// TIA Portal V17 export
// export: Created 2025-03-07T09:19:10.1766276Z, ExportSetting WithDefaults, DisplayName Totally Integrated Automation Portal, DisplayVersion V17 Update 8, DisplayName TIA Portal Openness, DisplayVersion V17 Update 8, DisplayName TIA Portal Version Control Interface, DisplayVersion V17, DisplayName SINAMICS Startdrive Advanced, DisplayVersion V17 SP2, DisplayName SINAMICS Startdrive G110M, G120, G120C, G120D, G120P, G115D, DisplayVersion V17 SP2, DisplayName SINAMICS Startdrive G130, G150, S120, S150, SINAMICS MV, S210, DisplayVersion V17 SP2, DisplayName STEP 7 Professional, DisplayVersion V17 Update 8, DisplayName SINUMERIK ONE STEP 7 Toolbox, DisplayVersion V17 Update 12, DisplayName SINUMERIK 840D sl STEP 7 Toolbox, DisplayVersion V17 Update 12, DisplayName STEP 7 Safety, DisplayVersion V17 Update 6, DisplayName WinCC Advanced, DisplayVersion V17 Update 8
FUNCTION "FC7216_RECIPES" : Void   // FC7216, LAD
{ S7_Optimized_Access := 'FALSE' }
AUTHOR : ETXETAR
VERSION : 1.0
// stored: AutoNumber false, IsIECCheckEnabled false, SetENOAutomatically false, UDAEnableTagReadback false
   VAR_TEMP
      STRING_AUX : String[254];
      TEMP0 : Int;
      NUM_OF_RECIPES : Int;
   END_VAR
   VAR CONSTANT
      FC_NUMBER : DInt := 7216;
   END_VAR
   VAR_TEMP   // added for the SCL form of the ladder/FBD networks
      _w1 : Bool;
      _w2 : Bool;
      _w3 : Bool;
   END_VAR
BEGIN

REGION Network 1: SEQUENCE IN PROCESS
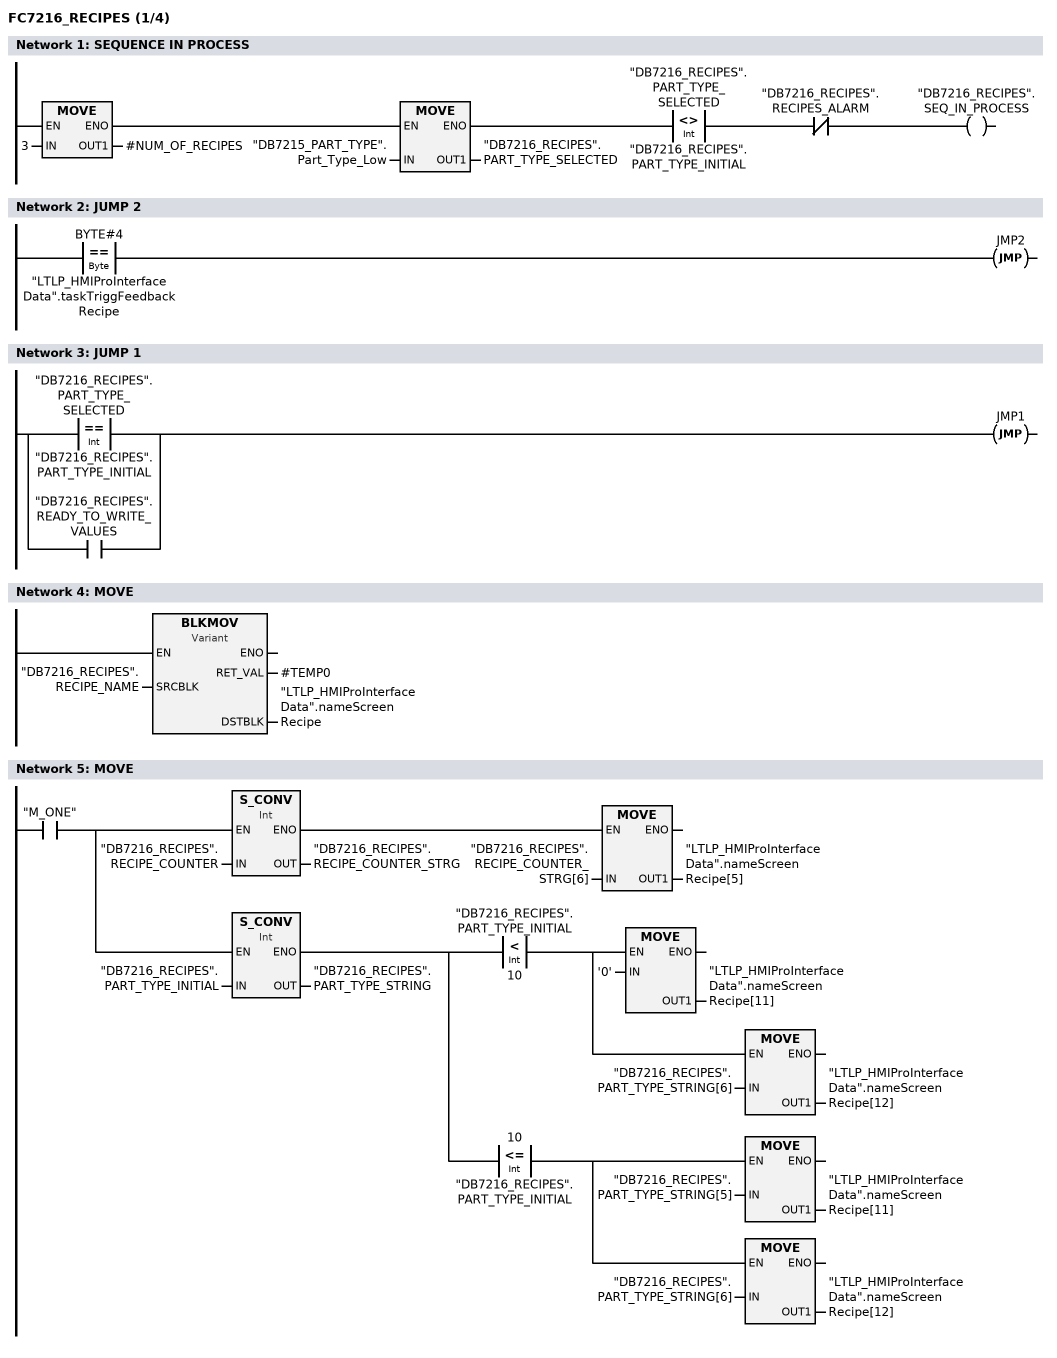
   RUNG wire#powerrail
      { S7_GenerateENO := "TRUE" } Move(in := 3, out1 => #NUM_OF_RECIPES)
      { S7_GenerateENO := "TRUE" } Move(in := "DB7215_PART_TYPE".Part_Type_Low, out1 => "DB7216_RECIPES".PART_TYPE_SELECTED)
      { S7_Templates := "SrcType := Int" } NE_Contact(in1 := "DB7216_RECIPES".PART_TYPE_SELECTED, in2 := "DB7216_RECIPES".PART_TYPE_INITIAL)
      I_Contact( "DB7216_RECIPES".RECIPES_ALARM )
      Coil( "DB7216_RECIPES".SEQ_IN_PROCESS )
   END_RUNG
   // the same network as SCL:
   // ENO of a box is taken as its EN; it also drops when the box reports an error
   #NUM_OF_RECIPES := 3;
   "DB7216_RECIPES".PART_TYPE_SELECTED := "DB7215_PART_TYPE".Part_Type_Low;
   "DB7216_RECIPES".SEQ_IN_PROCESS := ("DB7216_RECIPES".PART_TYPE_SELECTED <> "DB7216_RECIPES".PART_TYPE_INITIAL) AND NOT "DB7216_RECIPES".RECIPES_ALARM;
END_REGION

REGION Network 2: JUMP 2
   RUNG wire#powerrail
      { S7_Templates := "SrcType := Byte" } EQ_Contact(in1 := BYTE#4, in2 := "LTLP_HMIProInterfaceData".taskTriggFeedbackRecipe)
      JumpCoil( JMP2 )
   END_RUNG
   // the same network as SCL:
   IF BYTE#4 = "LTLP_HMIProInterfaceData".taskTriggFeedbackRecipe THEN GOTO JMP2; END_IF;
END_REGION

REGION Network 3: JUMP 1
   RUNG wire#powerrail
      { S7_Templates := "SrcType := Int" } EQ_Contact(in1 := "DB7216_RECIPES".PART_TYPE_SELECTED, in2 := "DB7216_RECIPES".PART_TYPE_INITIAL)
      wire#w1
      JumpCoil( JMP1 )
   END_RUNG
   RUNG wire#powerrail
      Contact( "DB7216_RECIPES".READY_TO_WRITE_VALUES )
   END_RUNG wire#w1
   // the same network as SCL:
   IF ("DB7216_RECIPES".PART_TYPE_SELECTED = "DB7216_RECIPES".PART_TYPE_INITIAL) OR "DB7216_RECIPES".READY_TO_WRITE_VALUES THEN
       GOTO JMP1;
   END_IF;
END_REGION

REGION Network 4: MOVE
   RUNG wire#powerrail
      { S7_Templates := "blk_type := Variant" } BLKMOV(SRCBLK := "DB7216_RECIPES".RECIPE_NAME, RET_VAL => #TEMP0, DSTBLK => "LTLP_HMIProInterfaceData".nameScreenRecipe)
   END_RUNG
   // the same network as SCL:
   #TEMP0 := BLKMOV(SRCBLK := "DB7216_RECIPES".RECIPE_NAME,
                    DSTBLK => "LTLP_HMIProInterfaceData".nameScreenRecipe);
END_REGION

REGION Network 5: MOVE
   RUNG wire#powerrail
      Contact( "M_ONE" )
      wire#w1
      { S7_Templates := "[src_type := Int, dest_type := String]" } S_CONV(IN := "DB7216_RECIPES".RECIPE_COUNTER, OUT => "DB7216_RECIPES".RECIPE_COUNTER_STRG)
      { S7_GenerateENO := "TRUE" } Move(in := "DB7216_RECIPES".RECIPE_COUNTER_STRG[6], out1 => "LTLP_HMIProInterfaceData".nameScreenRecipe[5])
   END_RUNG
   RUNG wire#w1
      { S7_Templates := "[src_type := Int, dest_type := String]" } S_CONV(IN := "DB7216_RECIPES".PART_TYPE_INITIAL, OUT => "DB7216_RECIPES".PART_TYPE_STRING)
      wire#w2
      { S7_Templates := "SrcType := Int" } LT_Contact(in1 := "DB7216_RECIPES".PART_TYPE_INITIAL, in2 := 10)
      wire#w3
      { S7_GenerateENO := "TRUE" } Move(in := '0', out1 => "LTLP_HMIProInterfaceData".nameScreenRecipe[11])
   END_RUNG
   RUNG wire#w3
      { S7_GenerateENO := "TRUE" } Move(in := "DB7216_RECIPES".PART_TYPE_STRING[6], out1 => "LTLP_HMIProInterfaceData".nameScreenRecipe[12])
   END_RUNG
   RUNG wire#w2
      { S7_Templates := "SrcType := Int" } LE_Contact(in1 := 10, in2 := "DB7216_RECIPES".PART_TYPE_INITIAL)
      wire#w4
      { S7_GenerateENO := "TRUE" } Move(in := "DB7216_RECIPES".PART_TYPE_STRING[5], out1 => "LTLP_HMIProInterfaceData".nameScreenRecipe[11])
   END_RUNG
   RUNG wire#w4
      { S7_GenerateENO := "TRUE" } Move(in := "DB7216_RECIPES".PART_TYPE_STRING[6], out1 => "LTLP_HMIProInterfaceData".nameScreenRecipe[12])
   END_RUNG
   // the same network as SCL:
   #_w2 := "M_ONE";
   S_CONV(EN := "M_ONE",
          IN := "DB7216_RECIPES".RECIPE_COUNTER,
          OUT => "DB7216_RECIPES".RECIPE_COUNTER_STRG,
          ENO => #_w1);
   IF #_w1 THEN
       "LTLP_HMIProInterfaceData".nameScreenRecipe[5] := "DB7216_RECIPES".RECIPE_COUNTER_STRG[6];
   END_IF;
   S_CONV(EN := #_w2,
          IN := "DB7216_RECIPES".PART_TYPE_INITIAL,
          OUT => "DB7216_RECIPES".PART_TYPE_STRING,
          ENO => #_w3);
   IF #_w3 AND ("DB7216_RECIPES".PART_TYPE_INITIAL < 10) THEN
       "LTLP_HMIProInterfaceData".nameScreenRecipe[11] := '0';
       "LTLP_HMIProInterfaceData".nameScreenRecipe[12] := "DB7216_RECIPES".PART_TYPE_STRING[6];
   END_IF;
   IF #_w3 AND (10 <= "DB7216_RECIPES".PART_TYPE_INITIAL) THEN
       "LTLP_HMIProInterfaceData".nameScreenRecipe[11] := "DB7216_RECIPES".PART_TYPE_STRING[5];
       "LTLP_HMIProInterfaceData".nameScreenRecipe[12] := "DB7216_RECIPES".PART_TYPE_STRING[6];
   END_IF;
END_REGION

REGION Network 6: MOVE
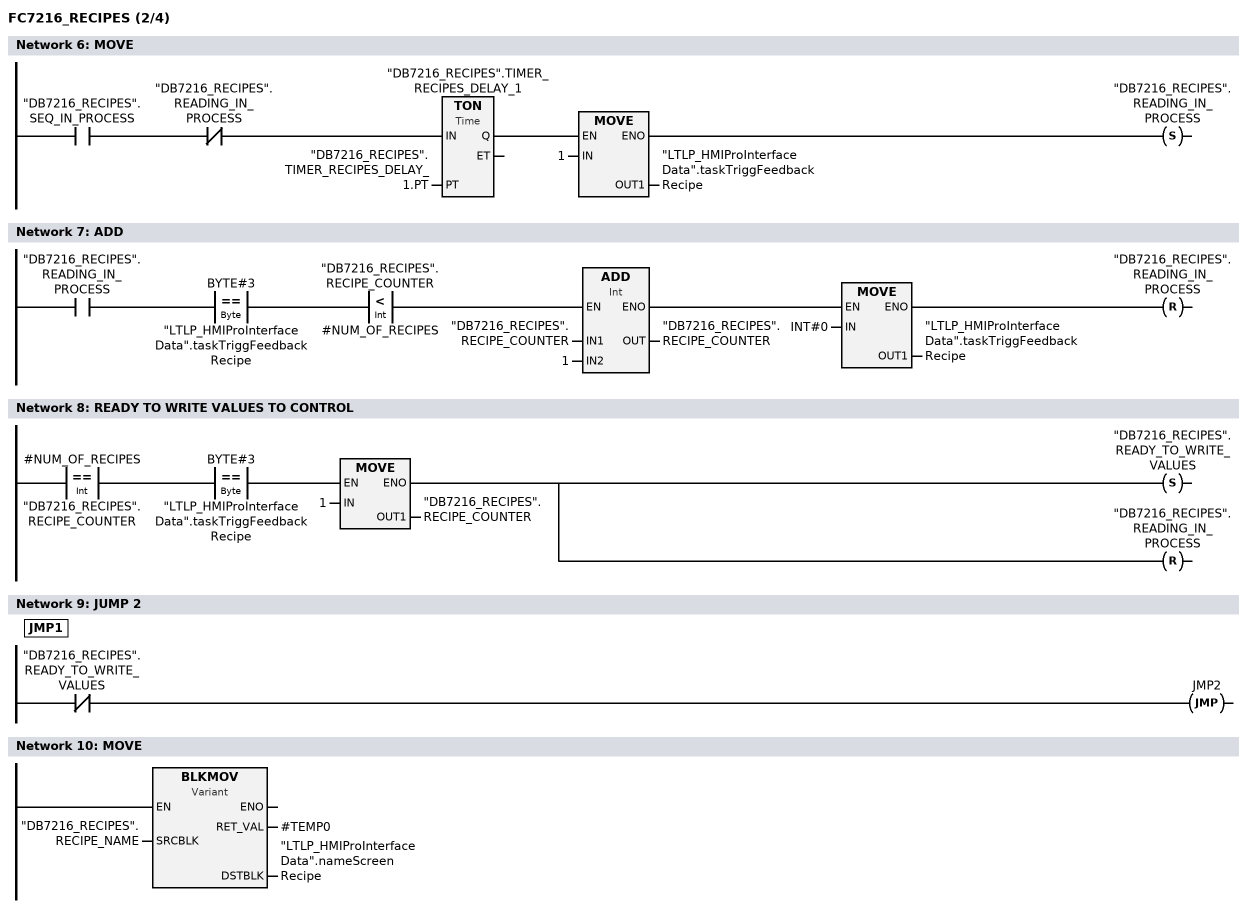
   RUNG wire#powerrail
      Contact( "DB7216_RECIPES".SEQ_IN_PROCESS )
      I_Contact( "DB7216_RECIPES".READING_IN_PROCESS )
      { S7_Templates := "time_type := Time" } "DB7216_RECIPES".TIMER_RECIPES_DELAY_1.TON(pt := "DB7216_RECIPES".TIMER_RECIPES_DELAY_1.PT, et =>)
      { S7_GenerateENO := "TRUE" } Move(in := 1, out1 => "LTLP_HMIProInterfaceData".taskTriggFeedbackRecipe)
      S_Coil( "DB7216_RECIPES".READING_IN_PROCESS )
   END_RUNG
   // the same network as SCL:
   // ENO of a box is taken as its EN; it also drops when the box reports an error
   "DB7216_RECIPES".TIMER_RECIPES_DELAY_1.TON(IN := "DB7216_RECIPES".SEQ_IN_PROCESS AND NOT "DB7216_RECIPES".READING_IN_PROCESS,
                           PT := "DB7216_RECIPES".TIMER_RECIPES_DELAY_1.PT);
   IF "DB7216_RECIPES".TIMER_RECIPES_DELAY_1.Q THEN
       "LTLP_HMIProInterfaceData".taskTriggFeedbackRecipe := 1;
       "DB7216_RECIPES".READING_IN_PROCESS := TRUE;
   END_IF;
END_REGION

REGION Network 7: ADD
   RUNG wire#powerrail
      Contact( "DB7216_RECIPES".READING_IN_PROCESS )
      { S7_Templates := "SrcType := Byte" } EQ_Contact(in1 := BYTE#3, in2 := "LTLP_HMIProInterfaceData".taskTriggFeedbackRecipe)
      { S7_Templates := "SrcType := Int" } LT_Contact(in1 := "DB7216_RECIPES".RECIPE_COUNTER, in2 := #NUM_OF_RECIPES)
      { S7_Templates := "SrcType := Int"; S7_GenerateENO := "TRUE" } Add(in1 := "DB7216_RECIPES".RECIPE_COUNTER, in2 := 1, out => "DB7216_RECIPES".RECIPE_COUNTER)
      { S7_GenerateENO := "TRUE" } Move(in := INT#0, out1 => "LTLP_HMIProInterfaceData".taskTriggFeedbackRecipe)
      R_Coil( "DB7216_RECIPES".READING_IN_PROCESS )
   END_RUNG
   // the same network as SCL:
   // ENO of a box is taken as its EN; it also drops when the box reports an error
   #_w1 := "DB7216_RECIPES".READING_IN_PROCESS AND (BYTE#3 = "LTLP_HMIProInterfaceData".taskTriggFeedbackRecipe) AND ("DB7216_RECIPES".RECIPE_COUNTER < #NUM_OF_RECIPES);
   IF #_w1 THEN
       "DB7216_RECIPES".RECIPE_COUNTER := "DB7216_RECIPES".RECIPE_COUNTER + 1;
       "LTLP_HMIProInterfaceData".taskTriggFeedbackRecipe := INT#0;
       "DB7216_RECIPES".READING_IN_PROCESS := FALSE;
   END_IF;
END_REGION

REGION Network 8: READY TO WRITE VALUES TO CONTROL
   RUNG wire#powerrail
      { S7_Templates := "SrcType := Int" } EQ_Contact(in1 := #NUM_OF_RECIPES, in2 := "DB7216_RECIPES".RECIPE_COUNTER)
      { S7_Templates := "SrcType := Byte" } EQ_Contact(in1 := BYTE#3, in2 := "LTLP_HMIProInterfaceData".taskTriggFeedbackRecipe)
      { S7_GenerateENO := "TRUE" } Move(in := 1, out1 => "DB7216_RECIPES".RECIPE_COUNTER)
      wire#w1
      S_Coil( "DB7216_RECIPES".READY_TO_WRITE_VALUES )
   END_RUNG
   RUNG wire#w1
      R_Coil( "DB7216_RECIPES".READING_IN_PROCESS )
   END_RUNG
   // the same network as SCL:
   // ENO of a box is taken as its EN; it also drops when the box reports an error
   #_w1 := (#NUM_OF_RECIPES = "DB7216_RECIPES".RECIPE_COUNTER) AND (BYTE#3 = "LTLP_HMIProInterfaceData".taskTriggFeedbackRecipe);
   IF #_w1 THEN
       "DB7216_RECIPES".RECIPE_COUNTER := 1;
       "DB7216_RECIPES".READY_TO_WRITE_VALUES := TRUE;
       "DB7216_RECIPES".READING_IN_PROCESS := FALSE;
   END_IF;
END_REGION

REGION Network 9: JUMP 2
   Label( JMP1 )
   RUNG wire#powerrail
      I_Contact( "DB7216_RECIPES".READY_TO_WRITE_VALUES )
      JumpCoil( JMP2 )
   END_RUNG
   // the same network as SCL:
   JMP1:
   IF NOT "DB7216_RECIPES".READY_TO_WRITE_VALUES THEN GOTO JMP2; END_IF;
END_REGION

REGION Network 10: MOVE
   RUNG wire#powerrail
      { S7_Templates := "blk_type := Variant" } BLKMOV(SRCBLK := "DB7216_RECIPES".RECIPE_NAME, RET_VAL => #TEMP0, DSTBLK => "LTLP_HMIProInterfaceData".nameScreenRecipe)
   END_RUNG
   // the same network as SCL:
   #TEMP0 := BLKMOV(SRCBLK := "DB7216_RECIPES".RECIPE_NAME,
                    DSTBLK => "LTLP_HMIProInterfaceData".nameScreenRecipe);
END_REGION

REGION Network 11: MOVE
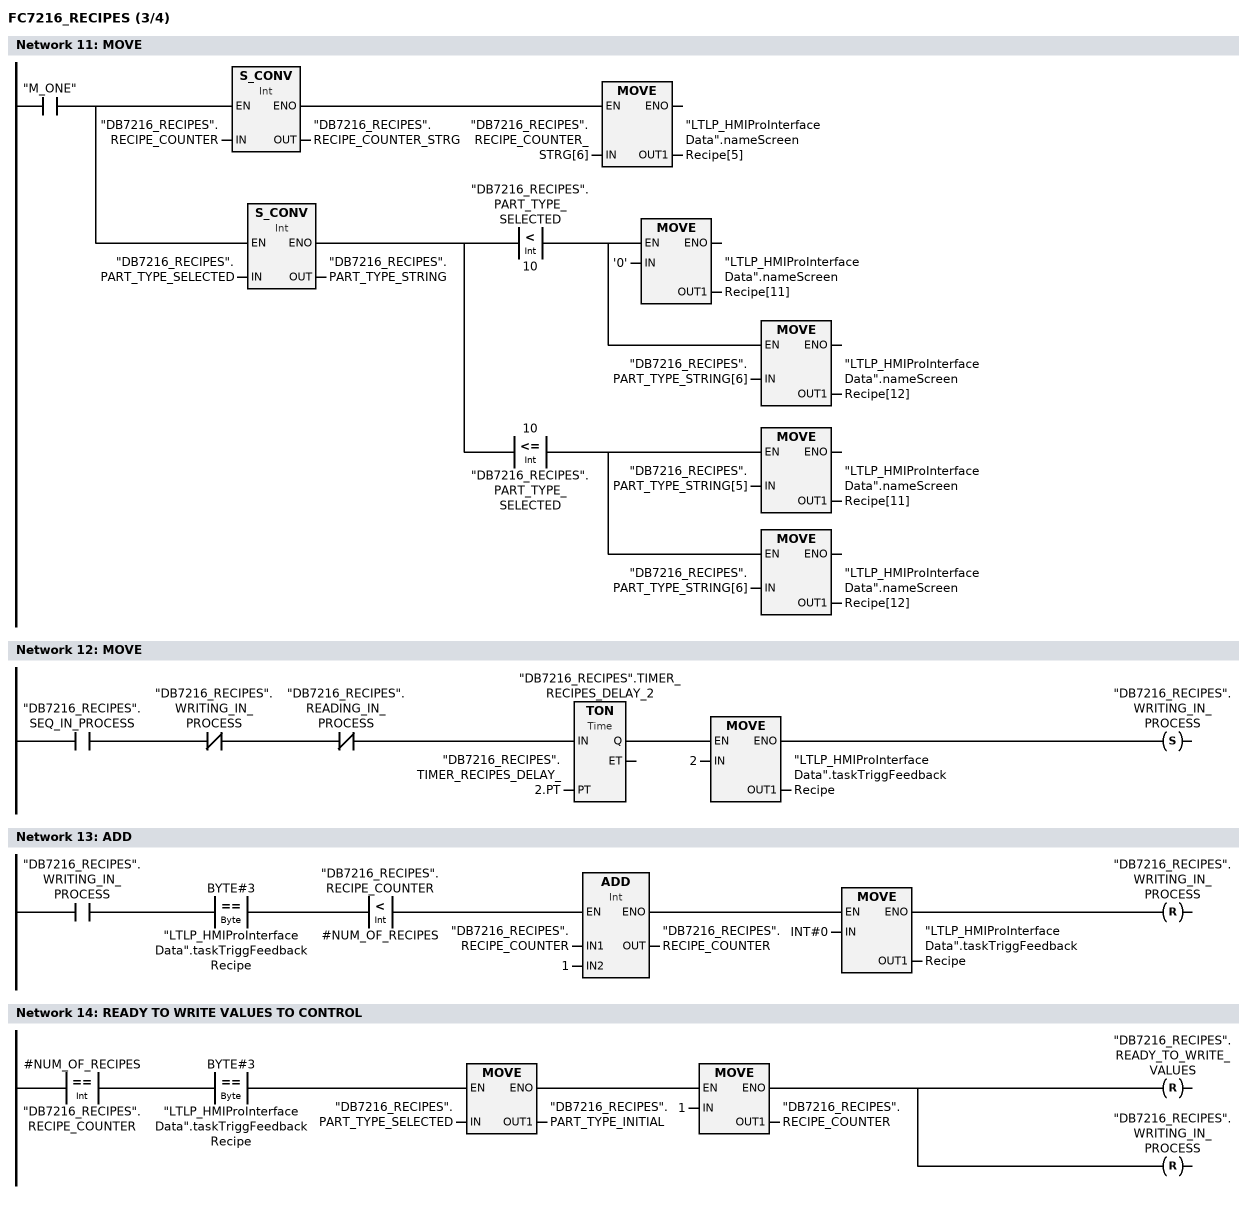
   RUNG wire#powerrail
      Contact( "M_ONE" )
      wire#w1
      { S7_Templates := "[src_type := Int, dest_type := String]" } S_CONV(IN := "DB7216_RECIPES".RECIPE_COUNTER, OUT => "DB7216_RECIPES".RECIPE_COUNTER_STRG)
      { S7_GenerateENO := "TRUE" } Move(in := "DB7216_RECIPES".RECIPE_COUNTER_STRG[6], out1 => "LTLP_HMIProInterfaceData".nameScreenRecipe[5])
   END_RUNG
   RUNG wire#w1
      { S7_Templates := "[src_type := Int, dest_type := String]" } S_CONV(IN := "DB7216_RECIPES".PART_TYPE_SELECTED, OUT => "DB7216_RECIPES".PART_TYPE_STRING)
      wire#w2
      { S7_Templates := "SrcType := Int" } LT_Contact(in1 := "DB7216_RECIPES".PART_TYPE_SELECTED, in2 := 10)
      wire#w3
      { S7_GenerateENO := "TRUE" } Move(in := '0', out1 => "LTLP_HMIProInterfaceData".nameScreenRecipe[11])
   END_RUNG
   RUNG wire#w3
      { S7_GenerateENO := "TRUE" } Move(in := "DB7216_RECIPES".PART_TYPE_STRING[6], out1 => "LTLP_HMIProInterfaceData".nameScreenRecipe[12])
   END_RUNG
   RUNG wire#w2
      { S7_Templates := "SrcType := Int" } LE_Contact(in1 := 10, in2 := "DB7216_RECIPES".PART_TYPE_SELECTED)
      wire#w4
      { S7_GenerateENO := "TRUE" } Move(in := "DB7216_RECIPES".PART_TYPE_STRING[5], out1 => "LTLP_HMIProInterfaceData".nameScreenRecipe[11])
   END_RUNG
   RUNG wire#w4
      { S7_GenerateENO := "TRUE" } Move(in := "DB7216_RECIPES".PART_TYPE_STRING[6], out1 => "LTLP_HMIProInterfaceData".nameScreenRecipe[12])
   END_RUNG
   // the same network as SCL:
   #_w2 := "M_ONE";
   S_CONV(EN := "M_ONE",
          IN := "DB7216_RECIPES".RECIPE_COUNTER,
          OUT => "DB7216_RECIPES".RECIPE_COUNTER_STRG,
          ENO => #_w1);
   IF #_w1 THEN
       "LTLP_HMIProInterfaceData".nameScreenRecipe[5] := "DB7216_RECIPES".RECIPE_COUNTER_STRG[6];
   END_IF;
   S_CONV(EN := #_w2,
          IN := "DB7216_RECIPES".PART_TYPE_SELECTED,
          OUT => "DB7216_RECIPES".PART_TYPE_STRING,
          ENO => #_w3);
   IF #_w3 AND ("DB7216_RECIPES".PART_TYPE_SELECTED < 10) THEN
       "LTLP_HMIProInterfaceData".nameScreenRecipe[11] := '0';
       "LTLP_HMIProInterfaceData".nameScreenRecipe[12] := "DB7216_RECIPES".PART_TYPE_STRING[6];
   END_IF;
   IF #_w3 AND (10 <= "DB7216_RECIPES".PART_TYPE_SELECTED) THEN
       "LTLP_HMIProInterfaceData".nameScreenRecipe[11] := "DB7216_RECIPES".PART_TYPE_STRING[5];
       "LTLP_HMIProInterfaceData".nameScreenRecipe[12] := "DB7216_RECIPES".PART_TYPE_STRING[6];
   END_IF;
END_REGION

REGION Network 12: MOVE
   RUNG wire#powerrail
      Contact( "DB7216_RECIPES".SEQ_IN_PROCESS )
      I_Contact( "DB7216_RECIPES".WRITING_IN_PROCESS )
      I_Contact( "DB7216_RECIPES".READING_IN_PROCESS )
      { S7_Templates := "time_type := Time" } "DB7216_RECIPES".TIMER_RECIPES_DELAY_2.TON(pt := "DB7216_RECIPES".TIMER_RECIPES_DELAY_2.PT, et =>)
      { S7_GenerateENO := "TRUE" } Move(in := 2, out1 => "LTLP_HMIProInterfaceData".taskTriggFeedbackRecipe)
      S_Coil( "DB7216_RECIPES".WRITING_IN_PROCESS )
   END_RUNG
   // the same network as SCL:
   // ENO of a box is taken as its EN; it also drops when the box reports an error
   "DB7216_RECIPES".TIMER_RECIPES_DELAY_2.TON(IN := "DB7216_RECIPES".SEQ_IN_PROCESS AND NOT "DB7216_RECIPES".WRITING_IN_PROCESS AND NOT "DB7216_RECIPES".READING_IN_PROCESS,
                           PT := "DB7216_RECIPES".TIMER_RECIPES_DELAY_2.PT);
   IF "DB7216_RECIPES".TIMER_RECIPES_DELAY_2.Q THEN
       "LTLP_HMIProInterfaceData".taskTriggFeedbackRecipe := 2;
       "DB7216_RECIPES".WRITING_IN_PROCESS := TRUE;
   END_IF;
END_REGION

REGION Network 13: ADD
   RUNG wire#powerrail
      Contact( "DB7216_RECIPES".WRITING_IN_PROCESS )
      { S7_Templates := "SrcType := Byte" } EQ_Contact(in1 := BYTE#3, in2 := "LTLP_HMIProInterfaceData".taskTriggFeedbackRecipe)
      { S7_Templates := "SrcType := Int" } LT_Contact(in1 := "DB7216_RECIPES".RECIPE_COUNTER, in2 := #NUM_OF_RECIPES)
      { S7_Templates := "SrcType := Int"; S7_GenerateENO := "TRUE" } Add(in1 := "DB7216_RECIPES".RECIPE_COUNTER, in2 := 1, out => "DB7216_RECIPES".RECIPE_COUNTER)
      { S7_GenerateENO := "TRUE" } Move(in := INT#0, out1 => "LTLP_HMIProInterfaceData".taskTriggFeedbackRecipe)
      R_Coil( "DB7216_RECIPES".WRITING_IN_PROCESS )
   END_RUNG
   // the same network as SCL:
   // ENO of a box is taken as its EN; it also drops when the box reports an error
   #_w1 := "DB7216_RECIPES".WRITING_IN_PROCESS AND (BYTE#3 = "LTLP_HMIProInterfaceData".taskTriggFeedbackRecipe) AND ("DB7216_RECIPES".RECIPE_COUNTER < #NUM_OF_RECIPES);
   IF #_w1 THEN
       "DB7216_RECIPES".RECIPE_COUNTER := "DB7216_RECIPES".RECIPE_COUNTER + 1;
       "LTLP_HMIProInterfaceData".taskTriggFeedbackRecipe := INT#0;
       "DB7216_RECIPES".WRITING_IN_PROCESS := FALSE;
   END_IF;
END_REGION

REGION Network 14: READY TO WRITE VALUES TO CONTROL
   RUNG wire#powerrail
      { S7_Templates := "SrcType := Int" } EQ_Contact(in1 := #NUM_OF_RECIPES, in2 := "DB7216_RECIPES".RECIPE_COUNTER)
      { S7_Templates := "SrcType := Byte" } EQ_Contact(in1 := BYTE#3, in2 := "LTLP_HMIProInterfaceData".taskTriggFeedbackRecipe)
      { S7_GenerateENO := "TRUE" } Move(in := "DB7216_RECIPES".PART_TYPE_SELECTED, out1 => "DB7216_RECIPES".PART_TYPE_INITIAL)
      { S7_GenerateENO := "TRUE" } Move(in := 1, out1 => "DB7216_RECIPES".RECIPE_COUNTER)
      wire#w1
      R_Coil( "DB7216_RECIPES".READY_TO_WRITE_VALUES )
   END_RUNG
   RUNG wire#w1
      R_Coil( "DB7216_RECIPES".WRITING_IN_PROCESS )
   END_RUNG
   // the same network as SCL:
   // ENO of a box is taken as its EN; it also drops when the box reports an error
   IF (#NUM_OF_RECIPES = "DB7216_RECIPES".RECIPE_COUNTER) AND (BYTE#3 = "LTLP_HMIProInterfaceData".taskTriggFeedbackRecipe) THEN
       "DB7216_RECIPES".PART_TYPE_INITIAL := "DB7216_RECIPES".PART_TYPE_SELECTED;
   END_IF;
   #_w1 := (#NUM_OF_RECIPES = "DB7216_RECIPES".RECIPE_COUNTER) AND (BYTE#3 = "LTLP_HMIProInterfaceData".taskTriggFeedbackRecipe);
   IF #_w1 THEN
       "DB7216_RECIPES".RECIPE_COUNTER := 1;
       "DB7216_RECIPES".READY_TO_WRITE_VALUES := FALSE;
       "DB7216_RECIPES".WRITING_IN_PROCESS := FALSE;
   END_IF;
END_REGION

REGION Network 15: READY TO WRITE VALUES TO CONTROL
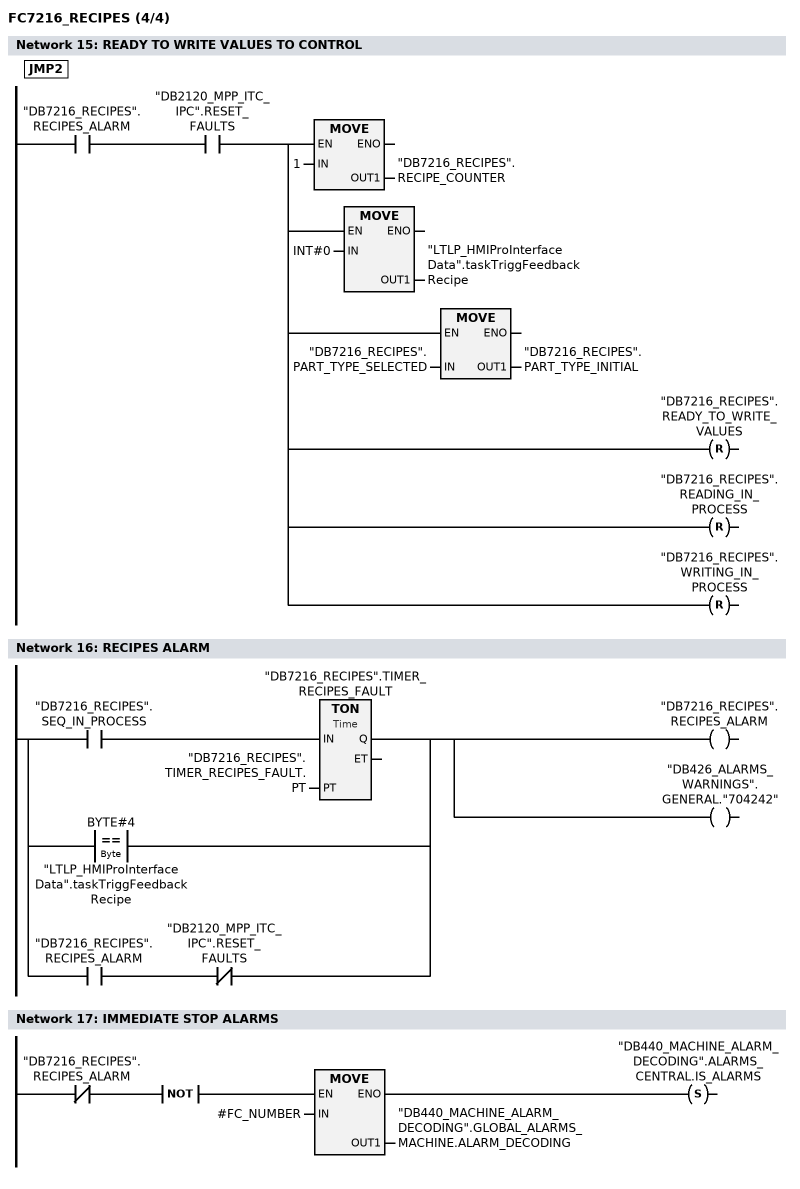
   Label( JMP2 )
   RUNG wire#powerrail
      Contact( "DB7216_RECIPES".RECIPES_ALARM )
      Contact( "DB2120_MPP_ITC_IPC".RESET_FAULTS )
      wire#w1
      { S7_GenerateENO := "TRUE" } Move(in := 1, out1 => "DB7216_RECIPES".RECIPE_COUNTER)
   END_RUNG
   RUNG wire#w1
      { S7_GenerateENO := "TRUE" } Move(in := INT#0, out1 => "LTLP_HMIProInterfaceData".taskTriggFeedbackRecipe)
   END_RUNG
   RUNG wire#w1
      { S7_GenerateENO := "TRUE" } Move(in := "DB7216_RECIPES".PART_TYPE_SELECTED, out1 => "DB7216_RECIPES".PART_TYPE_INITIAL)
   END_RUNG
   RUNG wire#w1
      R_Coil( "DB7216_RECIPES".READY_TO_WRITE_VALUES )
   END_RUNG
   RUNG wire#w1
      R_Coil( "DB7216_RECIPES".READING_IN_PROCESS )
   END_RUNG
   RUNG wire#w1
      R_Coil( "DB7216_RECIPES".WRITING_IN_PROCESS )
   END_RUNG
   // the same network as SCL:
   JMP2:
   IF "DB7216_RECIPES".RECIPES_ALARM AND "DB2120_MPP_ITC_IPC".RESET_FAULTS THEN
       "DB7216_RECIPES".RECIPE_COUNTER := 1;
       "LTLP_HMIProInterfaceData".taskTriggFeedbackRecipe := INT#0;
       "DB7216_RECIPES".PART_TYPE_INITIAL := "DB7216_RECIPES".PART_TYPE_SELECTED;
       "DB7216_RECIPES".READY_TO_WRITE_VALUES := FALSE;
       "DB7216_RECIPES".READING_IN_PROCESS := FALSE;
       "DB7216_RECIPES".WRITING_IN_PROCESS := FALSE;
   END_IF;
END_REGION

REGION Network 16: RECIPES ALARM
   RUNG wire#powerrail
      Contact( "DB7216_RECIPES".SEQ_IN_PROCESS )
      { S7_Templates := "time_type := Time" } "DB7216_RECIPES".TIMER_RECIPES_FAULT.TON(pt := "DB7216_RECIPES".TIMER_RECIPES_FAULT.PT, et =>)
      wire#w1
      Coil( "DB7216_RECIPES".RECIPES_ALARM )
   END_RUNG
   RUNG wire#powerrail
      { S7_Templates := "SrcType := Byte" } EQ_Contact(in1 := BYTE#4, in2 := "LTLP_HMIProInterfaceData".taskTriggFeedbackRecipe)
   END_RUNG wire#w1
   RUNG wire#powerrail
      Contact( "DB7216_RECIPES".RECIPES_ALARM )
      I_Contact( "DB2120_MPP_ITC_IPC".RESET_FAULTS )
   END_RUNG wire#w1
   RUNG wire#w1
      Coil( "DB426_ALARMS_WARNINGS".GENERAL."704242" )
   END_RUNG
   // the same network as SCL:
   "DB7216_RECIPES".TIMER_RECIPES_FAULT.TON(IN := "DB7216_RECIPES".SEQ_IN_PROCESS,
                           PT := "DB7216_RECIPES".TIMER_RECIPES_FAULT.PT);
   "DB7216_RECIPES".RECIPES_ALARM := "DB7216_RECIPES".TIMER_RECIPES_FAULT.Q OR (BYTE#4 = "LTLP_HMIProInterfaceData".taskTriggFeedbackRecipe) OR ("DB7216_RECIPES".RECIPES_ALARM AND NOT "DB2120_MPP_ITC_IPC".RESET_FAULTS);
   "DB426_ALARMS_WARNINGS".GENERAL."704242" := "DB7216_RECIPES".RECIPES_ALARM;
END_REGION

REGION Network 17: IMMEDIATE STOP ALARMS
   RUNG wire#powerrail
      I_Contact( "DB7216_RECIPES".RECIPES_ALARM )
      Not()
      { S7_GenerateENO := "TRUE" } Move(in := #FC_NUMBER, out1 => "DB440_MACHINE_ALARM_DECODING".GLOBAL_ALARMS_MACHINE.ALARM_DECODING)
      S_Coil( "DB440_MACHINE_ALARM_DECODING".ALARMS_CENTRAL.IS_ALARMS )
   END_RUNG
   // the same network as SCL:
   // ENO of a box is taken as its EN; it also drops when the box reports an error
   IF NOT (NOT "DB7216_RECIPES".RECIPES_ALARM) THEN
       "DB440_MACHINE_ALARM_DECODING".GLOBAL_ALARMS_MACHINE.ALARM_DECODING := #FC_NUMBER;
       "DB440_MACHINE_ALARM_DECODING".ALARMS_CENTRAL.IS_ALARMS := TRUE;
   END_IF;
END_REGION
END_FUNCTION
